PROGRAM MAIN
VAR

END_VAR


//valves
FEE_VGC_02(
	i_stUSG:= FEE_KMONO_GCC_01.IG, 
	i_stDSG:= FEE_KMONO_GCC_01.IG , 
	i_xDis_DPIlk:= FALSE, 
	i_xEPS_OK:= FALSE, 
	i_xPMPS_OK:= , 
	i_xExt_OK:= TRUE, 
	i_xOverrideMode:= , 
	i_xReset:= , 
	iq_stValve=> , 
	xMPS_OK=> , 
	io_fbFFHWO:= g_FastFaultOutput1 );

FEE_VGC_03(
	i_stUSG:=FEE_KMONO_GCC_01.IG, 
	i_stDSG:= FEE_M1L_GCC_01.IG , 
	i_xDis_DPIlk:= FALSE, 
	i_xEPS_OK:= FALSE, 
	i_xPMPS_OK:= TRUE, 
	i_xExt_OK:= TRUE, 
	i_xOverrideMode:= , 
	i_xReset:= , 
	iq_stValve=> , 
	xMPS_OK=> , 
	io_fbFFHWO:= g_FastFaultOutput1 );

FEE_VGC_04(
	i_stUSG:= FEE_GCC_03.IG, 
	i_stDSG:= FEE_GCC_03.IG , 
	i_xDis_DPIlk:= FALSE, 
	i_xEPS_OK:= FALSE, 
	i_xPMPS_OK:= TRUE, 
	i_xExt_OK:= TRUE, 
	i_xOverrideMode:= , 
	i_xReset:= , 
	iq_stValve=> , 
	xMPS_OK=> , 
	io_fbFFHWO:= g_FastFaultOutput1 );	
	
// gauges and pip
FEE_KMONO_GPI_01(PG=>);
FEE_KMONO_GCC_01(PG:=FEE_KMONO_GPI_01.PG);
FEE_KMONO_PIP_01(i_stGauge:= FEE_KMONO_GCC_01.IG);

FEE_GPI_03(PG=>);
FEE_GCC_03(PG:=FEE_KMONO_GPI_01.PG);

FEE_PIP_02(i_stGauge:= FEE_GCC_03.IG);

FEE_M1L_GPI_01(PG=>);
FEE_M1L_GCC_01(PG:=FEE_M1L_GPI_01.PG);
FEE_M1L_PIP_01(i_stGauge:= FEE_M1L_GCC_01.IG);

FEE_GPI_04(PG=>);
FEE_GCC_04(PG:=FEE_GPI_04.PG);
FEE_PIP_03(i_stGauge:= FEE_GCC_04.IG);

END_PROGRAM

(* stored: Version 1.1.0.1, ProductVersion 3.1.4022.12
   POU MAIN: Id {a967ae7f-2447-4741-99c2-9f2a87c804ab}, SpecialFunc None *)
